{attribute 'GeneratedUsingTerminal: EL9210-0000-0016'}
{attribute addProperty BoxType "EL9210-0000-0016"}
{attribute addProperty Id "PowerOKAT %I*BOOL1"}
{attribute addProperty CRC "3467836690"}
{attribute addProperty Size "1"}
TYPE PowerOK_CEB2FD12 EXTENDS InputBase_8311D824 :
STRUCT
	{attribute addProperty Name "PowerOK"}
	PowerOK AT %I* : BOOL;
END_STRUCT
END_TYPE

(* stored: Version 1.2.0.0, ProductVersion 3.1.4024.9
   DUT PowerOK_CEB2FD12: Id {5cf8116b-5457-4fc8-9ed5-1ae820005eec} *)
